// TIA Portal V20 export
DATA_BLOCK "DB_CITI_ToolingMap"   // DB391
TITLE = GMPT Common Logic Data Block for I.T. Tooling Memory Map
AUTHOR : JRose
FAMILY : CITI
NAME : MMG3.2
VERSION : 0.0
// stored: MemoryReserve 0, Namespace CITI_Logic
   VAR RETAIN
      Tool : Array[1..140] of "CITI_Logic.zp_Tool_Data";
   END_VAR
BEGIN
END_DATA_BLOCK
